FUNCTION_BLOCK FB_PosTest
VAR_INPUT
	PosTargetR : DINT;
	PosTargetL : DINT;
END_VAR
VAR_OUTPUT
	ApplyPosTargetNow : BOOL :=FALSE;
	PosCmd : DINT;
	nCycles : DINT := 0;
END_VAR
VAR
	eStateMachine		: E_PosTest := E_PosTest.Idle_init;
	inWindow : BOOL := TRUE;
	waitApplyPosTargetNow : UDINT;
END_VAR

METHOD Execute : BOOL
VAR_INPUT
END_VAR
VAR
END_VAR
CASE eStateMachine OF
	E_PosTest.Idle_init:
		ApplyPosTargetNow := FALSE;
		waitApplyPosTargetNow:=1000;
		IF Ds402.StatusWord_Bits.SwitchOn THEN
			eStateMachine := E_PosTest.Idle_start;
		END_IF
	E_PosTest.Idle_start:
	waitApplyPosTargetNow:=waitApplyPosTargetNow-1;
	IF waitApplyPosTargetNow =0 THEN
		eStateMachine := E_PosTest.GoToNextState_levelHi;
	END_IF
	
	E_PosTest.GoToNextState_levelHi:
	nCycles:=nCycles+1;
		PosCmd := PosTargetR;
		ApplyPosTargetNow := TRUE;//waitApplyPosTargetNow:=1000;
		eStateMachine := E_PosTest.MovingTo_levelHi;
		inWindow := TRUE;
	E_PosTest.MovingTo_levelHi:
		//waitApplyPosTargetNow:=waitApplyPosTargetNow-1;
		//IF  waitApplyPosTargetNow=0  THEN
		//ApplyPosTargetNow := FALSE;
		//END_IF
			IF Ds402.StatusWord_Bits.SetPointAck THEN
				ApplyPosTargetNow := FALSE;
			END_IF

		IF NOT Ds402.StatusWord_Bits.TargetReached THEN
			inWindow := FALSE;
		END_IF
		IF  Ds402.StatusWord_Bits.TargetReached AND NOT inWindow THEN
			eStateMachine := E_PosTest.GoToNextState_levelLo;
		END_IF

	E_PosTest.GoToNextState_levelLo:
		PosCmd := PosTargetL;
		ApplyPosTargetNow := TRUE;//waitApplyPosTargetNow:=1000;
		eStateMachine := E_PosTest.MovingTo_levelLo;
		inWindow := TRUE;
	E_PosTest.MovingTo_levelLo:
		//waitApplyPosTargetNow:=waitApplyPosTargetNow-1;
		//IF  waitApplyPosTargetNow=0  THEN
		//	ApplyPosTargetNow := FALSE;
		//END_IF
		IF Ds402.StatusWord_Bits.SetPointAck THEN
			ApplyPosTargetNow := FALSE;
		END_IF

		IF NOT Ds402.StatusWord_Bits.TargetReached THEN
			inWindow := FALSE;
		END_IF
		IF  Ds402.StatusWord_Bits.TargetReached AND NOT inWindow THEN
			eStateMachine := E_PosTest.GoToNextState_levelHi;
		END_IF
		
END_CASE


ServoCtrl.PosTarget := PosCmd;
ServoCtrl.TargetTorque := 0;
ServoCtrl.ModeOfOperation := TO_SINT(E_ModesOfOperation.ED_MO_Profile_position_mode);
END_METHOD

METHOD Restart : BOOL
VAR_INPUT
END_VAR
	eStateMachine		  := E_PosTest.Idle_init;
	inWindow   := TRUE;
	nCycles    :=  0;
END_METHOD

END_FUNCTION_BLOCK

(* stored: Version 1.1.0.1, ProductVersion 3.1.4024.13
   POU FB_PosTest: Id {4aec3ffd-4b45-43d2-82c4-3567bfb43c10}, SpecialFunc None
   Method Execute: Id {1051fbff-c7f9-44ae-b67e-9bac046637ed}
   Method Restart: Id {723566c6-5b1e-4908-9f6f-22281a13a987} *)
